(* DUT: E_StudyState *)

TYPE E_StudyState :
(
    Idle,        (* no timer running *)
    Work,        (* working 25 min *)
    ShortBreak,  (* 5 min break *)
    LongBreak,   (* 15 min break *)
    Paused       (* paused during work *)
);
END_TYPE

(* stored: Version 1.1.0.1, ProductVersion 3.1.4024.16
   DUT E_StudyState: Id {1cd7fa6c-6b59-4647-831f-fd0218a865d0} *)
